TYPE Interpolation_FunctionResult :
(
	Interpolation_OK := -1,
	Interpolation_Busy := 0,
	Interpolation_Error,
	Interpolation_OutOfBounds,
	Interpolation_Assignment_Cannot_Be_Same,
	Interpolation_Aborted
);
END_TYPE

(* stored: Version 1.1.0.1, ProductVersion 3.1.4020.3
   DUT Interpolation_FunctionResult: Id {524dce41-f844-49f2-aef6-457ae50912a4} *)
